FUNCTION_BLOCK PUBLIC WORD_TO_TestSuite EXTENDS TcUnit.FB_TestSuite
VAR
END_VAR

Check_WORD_TO_BOOL_Max();
Check_WORD_TO_BOOL_Min();
Check_WORD_TO_BYTE_Max();
Check_WORD_TO_BYTE_Min();
Check_WORD_TO_BYTE_TooHigh();
Check_WORD_TO_WORD_Max();
Check_WORD_TO_WORD_Min();
Check_WORD_TO_DWORD_Max();
Check_WORD_TO_DWORD_Min();
Check_WORD_TO_LWORD_Max();
Check_WORD_TO_LWORD_Min();
Check_WORD_TO_SINT_Max();
Check_WORD_TO_SINT_Min();
Check_WORD_TO_SINT_TooHigh();
Check_WORD_TO_INT_Max();
Check_WORD_TO_INT_Min();
Check_WORD_TO_INT_TooHigh();
Check_WORD_TO_DINT_Max();
Check_WORD_TO_DINT_Min();
Check_WORD_TO_LINT_Max();
Check_WORD_TO_LINT_Min();
Check_WORD_TO_USINT_Max();
Check_WORD_TO_USINT_Min();
Check_WORD_TO_USINT_TooHigh();
Check_WORD_TO_UINT_Max();
Check_WORD_TO_UINT_Min();
Check_WORD_TO_UDINT_Max();
Check_WORD_TO_UDINT_Min();
Check_WORD_TO_ULINT_Max();
Check_WORD_TO_ULINT_Min();
Check_WORD_TO_REAL_Max();
Check_WORD_TO_REAL_Min();
Check_WORD_TO_LREAL_Max();
Check_WORD_TO_LREAL_Min();
Check_WORD_TO_TIME_Max();
Check_WORD_TO_TIME_Min();
Check_WORD_TO_TOD_Max();
Check_WORD_TO_TOD_Min();
Check_WORD_TO_DATE_Max();
Check_WORD_TO_DATE_Min();
Check_WORD_TO_DT_Max();
Check_WORD_TO_DT_Min();
Check_WORD_TO_STRING_Max();
Check_WORD_TO_STRING_Min();

METHOD PUBLIC Check_WORD_TO_BOOL_Min
VAR
	value : WORD := DatatypeLimits.WORD_MIN_VALUE;
	actual : BOOL;
	converted : BOOL;
	equal : BOOL;
END_VAR
TEST('Check_WORD_TO_BOOL_Min');

// @TEST-RUN
converted := TryConvert_WORD_TO_Destination(value, actual);
equal := actual = WORD_TO_BOOL(value);

// @TEST-ASSERT
AssertTrue(Condition := equal, Message := 'Did not convert WORD to BOOL correctly');
AssertTrue(Condition := converted, Message := 'Did not report WORD to BOOL conversion was successful');

TEST_FINISHED();
END_METHOD

METHOD PUBLIC Check_WORD_TO_BOOL_Max
VAR
	value : WORD := DatatypeLimits.WORD_MAX_VALUE;
	actual : BOOL;
	converted : BOOL;
	equal : BOOL;
END_VAR
TEST('Check_WORD_TO_BOOL_Max');

// @TEST-RUN
converted := TryConvert_WORD_TO_Destination(value, actual);
equal := actual = WORD_TO_BOOL(value);

// @TEST-ASSERT
AssertTrue(Condition := equal, Message := 'Did not convert WORD to BOOL correctly');
AssertTrue(Condition := converted, Message := 'Did not report WORD to BOOL conversion was successful');

TEST_FINISHED();
END_METHOD

METHOD PUBLIC Check_WORD_TO_BYTE_Min
VAR
	value : WORD := DatatypeLimits.WORD_MIN_VALUE;
	actual : BYTE;
	converted : BOOL;
	equal : BOOL;
END_VAR
TEST('Check_WORD_TO_BYTE_Min');

// @TEST-RUN
converted := TryConvert_WORD_TO_Destination(value, actual);
equal := actual = WORD_TO_BYTE(value);

// @TEST-ASSERT
AssertTrue(Condition := equal, Message := 'Did not convert WORD to BYTE correctly');
AssertTrue(Condition := converted, Message := 'Did not report WORD to BYTE conversion was successful');

TEST_FINISHED();
END_METHOD

METHOD PUBLIC Check_WORD_TO_BYTE_TooHigh
VAR
	value : WORD := DatatypeLimits.WORD_MAX_VALUE;
	actual : BYTE;
	converted : BOOL;
END_VAR
TEST('Check_WORD_TO_BYTE_TooHigh');

// @TEST-RUN
converted := TryConvert_WORD_TO_Destination(value, actual);

// @TEST-ASSERT
AssertFalse(Condition := converted, Message := 'Did not report WORD to BYTE conversion was prevented');

TEST_FINISHED();
END_METHOD

METHOD PUBLIC Check_WORD_TO_BYTE_Max
VAR
	value : WORD := DatatypeLimits.MAX_VALUE_OF_WORD_WHICH_CAN_BE_HELD_IN_A_BYTE;
	actual : BYTE;
	converted : BOOL;
	equal : BOOL;
END_VAR
TEST('Check_WORD_TO_BYTE_Max');

// @TEST-RUN
converted := TryConvert_WORD_TO_Destination(value, actual);
equal := actual = WORD_TO_BYTE(value);

// @TEST-ASSERT
AssertTrue(Condition := equal, Message := 'Did not convert WORD to BYTE correctly');
AssertTrue(Condition := converted, Message := 'Did not report WORD to BYTE conversion was successful');

TEST_FINISHED();
END_METHOD

METHOD PUBLIC Check_WORD_TO_DATE_Min
VAR
	value : WORD := DatatypeLimits.WORD_MIN_VALUE;
	actual : DATE;
	converted : BOOL;
	equal : BOOL;
END_VAR
TEST('Check_WORD_TO_DATE_Min');

// @TEST-RUN
converted := TryConvert_WORD_TO_Destination(value, actual);
equal := actual = WORD_TO_DATE(value);

// @TEST-ASSERT
AssertTrue(Condition := equal, Message := 'Did not convert WORD to DATE correctly');
AssertTrue(Condition := converted, Message := 'Did not report WORD to DATE conversion was successful');

TEST_FINISHED();
END_METHOD

METHOD PUBLIC Check_WORD_TO_DATE_Max
VAR
	value : WORD := DatatypeLimits.WORD_MAX_VALUE;
	actual : DATE;
	converted : BOOL;
	equal : BOOL;
END_VAR
TEST('Check_WORD_TO_DATE_Max');

// @TEST-RUN
converted := TryConvert_WORD_TO_Destination(value, actual);
equal := actual = WORD_TO_DATE(value);

// @TEST-ASSERT
AssertTrue(Condition := equal, Message := 'Did not convert WORD to DATE correctly');
AssertTrue(Condition := converted, Message := 'Did not report WORD to DATE conversion was successful');

TEST_FINISHED();
END_METHOD

METHOD PUBLIC Check_WORD_TO_DINT_Min
VAR
	value : WORD := DatatypeLimits.WORD_MIN_VALUE;
	actual : DINT;
	converted : BOOL;
	equal : BOOL;
END_VAR
TEST('Check_WORD_TO_DINT_Min');

// @TEST-RUN
converted := TryConvert_WORD_TO_Destination(value, actual);
equal := actual = WORD_TO_DINT(value);

// @TEST-ASSERT
AssertTrue(Condition := equal, Message := 'Did not convert WORD to DINT correctly');
AssertTrue(Condition := converted, Message := 'Did not report WORD to DINT conversion was successful');

TEST_FINISHED();
END_METHOD

METHOD PUBLIC Check_WORD_TO_DINT_Max
VAR
	value : WORD := DatatypeLimits.WORD_MAX_VALUE;
	actual : DINT;
	converted : BOOL;
	equal : BOOL;
END_VAR
TEST('Check_WORD_TO_DINT_Max');

// @TEST-RUN
converted := TryConvert_WORD_TO_Destination(value, actual);
equal := actual = WORD_TO_DINT(value);

// @TEST-ASSERT
AssertTrue(Condition := equal, Message := 'Did not convert WORD to DINT correctly');
AssertTrue(Condition := converted, Message := 'Did not report WORD to DINT conversion was successful');

TEST_FINISHED();
END_METHOD

METHOD PUBLIC Check_WORD_TO_DT_Min
VAR
	value : WORD := DatatypeLimits.WORD_MIN_VALUE;
	actual : DT;
	converted : BOOL;
	equal : BOOL;
END_VAR
TEST('Check_WORD_TO_DT_Min');

// @TEST-RUN
converted := TryConvert_WORD_TO_Destination(value, actual);
equal := actual = WORD_TO_DT(value);

// @TEST-ASSERT
AssertTrue(Condition := equal, Message := 'Did not convert WORD to DT correctly');
AssertTrue(Condition := converted, Message := 'Did not report WORD to DT conversion was successful');

TEST_FINISHED();
END_METHOD

METHOD PUBLIC Check_WORD_TO_DT_Max
VAR
	value : WORD := DatatypeLimits.WORD_MAX_VALUE;
	actual : DT;
	converted : BOOL;
	equal : BOOL;
END_VAR
TEST('Check_WORD_TO_DT_Max');

// @TEST-RUN
converted := TryConvert_WORD_TO_Destination(value, actual);
equal := actual = WORD_TO_DT(value);

// @TEST-ASSERT
AssertTrue(Condition := equal, Message := 'Did not convert WORD to DT correctly');
AssertTrue(Condition := converted, Message := 'Did not report WORD to DT conversion was successful');

TEST_FINISHED();
END_METHOD

METHOD PUBLIC Check_WORD_TO_DWORD_Min
VAR
	value : WORD := DatatypeLimits.WORD_MIN_VALUE;
	actual : DWORD;
	converted : BOOL;
	equal : BOOL;
END_VAR
TEST('Check_WORD_TO_DWORD_Min');

// @TEST-RUN
converted := TryConvert_WORD_TO_Destination(value, actual);
equal := actual = WORD_TO_DWORD(value);

// @TEST-ASSERT
AssertTrue(Condition := equal, Message := 'Did not convert WORD to DWORD correctly');
AssertTrue(Condition := converted, Message := 'Did not report WORD to DWORD conversion was successful');

TEST_FINISHED();
END_METHOD

METHOD PUBLIC Check_WORD_TO_DWORD_Max
VAR
	value : WORD := DatatypeLimits.WORD_MAX_VALUE;
	actual : DWORD;
	converted : BOOL;
	equal : BOOL;
END_VAR
TEST('Check_WORD_TO_DWORD_Max');

// @TEST-RUN
converted := TryConvert_WORD_TO_Destination(value, actual);
equal := actual = WORD_TO_DWORD(value);

// @TEST-ASSERT
AssertTrue(Condition := equal, Message := 'Did not convert WORD to DWORD correctly');
AssertTrue(Condition := converted, Message := 'Did not report WORD to DWORD conversion was successful');

TEST_FINISHED();
END_METHOD

METHOD PUBLIC Check_WORD_TO_INT_Min
VAR
	value : WORD := DatatypeLimits.WORD_MIN_VALUE;
	actual : INT;
	converted : BOOL;
	equal : BOOL;
END_VAR
TEST('Check_WORD_TO_INT_Min');

// @TEST-RUN
converted := TryConvert_WORD_TO_Destination(value, actual);
equal := actual = WORD_TO_INT(value);

// @TEST-ASSERT
AssertTrue(Condition := equal, Message := 'Did not convert WORD to INT correctly');
AssertTrue(Condition := converted, Message := 'Did not report WORD to INT conversion was successful');

TEST_FINISHED();
END_METHOD

METHOD PUBLIC Check_WORD_TO_INT_TooHigh
VAR
	value : WORD := DatatypeLimits.WORD_MAX_VALUE;
	actual : INT;
	converted : BOOL;
END_VAR
TEST('Check_WORD_TO_INT_TooHigh');

// @TEST-RUN
converted := TryConvert_WORD_TO_Destination(value, actual);

// @TEST-ASSERT
AssertFalse(Condition := converted, Message := 'Did not report WORD to INT conversion was prevented');

TEST_FINISHED();
END_METHOD

METHOD PUBLIC Check_WORD_TO_INT_Max
VAR
	value : WORD := DatatypeLimits.MAX_VALUE_OF_WORD_WHICH_CAN_BE_HELD_IN_A_INT;
	actual : INT;
	converted : BOOL;
	equal : BOOL;
END_VAR
TEST('Check_WORD_TO_INT_Max');

// @TEST-RUN
converted := TryConvert_WORD_TO_Destination(value, actual);
equal := actual = WORD_TO_INT(value);

// @TEST-ASSERT
AssertTrue(Condition := equal, Message := 'Did not convert WORD to INT correctly');
AssertTrue(Condition := converted, Message := 'Did not report WORD to INT conversion was successful');

TEST_FINISHED();
END_METHOD

METHOD PUBLIC Check_WORD_TO_LINT_Min
VAR
	value : WORD := DatatypeLimits.WORD_MIN_VALUE;
	actual : LINT;
	converted : BOOL;
	equal : BOOL;
END_VAR
TEST('Check_WORD_TO_LINT_Min');

// @TEST-RUN
converted := TryConvert_WORD_TO_Destination(value, actual);
equal := actual = WORD_TO_LINT(value);

// @TEST-ASSERT
AssertTrue(Condition := equal, Message := 'Did not convert WORD to LINT correctly');
AssertTrue(Condition := converted, Message := 'Did not report WORD to LINT conversion was successful');

TEST_FINISHED();
END_METHOD

METHOD PUBLIC Check_WORD_TO_LINT_Max
VAR
	value : WORD := DatatypeLimits.WORD_MAX_VALUE;
	actual : LINT;
	converted : BOOL;
	equal : BOOL;
END_VAR
TEST('Check_WORD_TO_LINT_Max');

// @TEST-RUN
converted := TryConvert_WORD_TO_Destination(value, actual);
equal := actual = WORD_TO_LINT(value);

// @TEST-ASSERT
AssertTrue(Condition := equal, Message := 'Did not convert WORD to LINT correctly');
AssertTrue(Condition := converted, Message := 'Did not report WORD to LINT conversion was successful');

TEST_FINISHED();
END_METHOD

METHOD PUBLIC Check_WORD_TO_LREAL_Min
VAR
	value : WORD := DatatypeLimits.WORD_MIN_VALUE;
	actual : LREAL;
	converted : BOOL;
	equal : BOOL;
END_VAR
TEST('Check_WORD_TO_LREAL_Min');

// @TEST-RUN
converted := TryConvert_WORD_TO_Destination(value, actual);
equal := actual = WORD_TO_LREAL(value);

// @TEST-ASSERT
AssertTrue(Condition := equal, Message := 'Did not convert WORD to LREAL correctly');
AssertTrue(Condition := converted, Message := 'Did not report WORD to LREAL conversion was successful');

TEST_FINISHED();
END_METHOD

METHOD PUBLIC Check_WORD_TO_LREAL_Max
VAR
	value : WORD := DatatypeLimits.WORD_MAX_VALUE;
	actual : LREAL;
	converted : BOOL;
	equal : BOOL;
END_VAR
TEST('Check_WORD_TO_LREAL_Max');

// @TEST-RUN
converted := TryConvert_WORD_TO_Destination(value, actual);
equal := actual = WORD_TO_LREAL(value);

// @TEST-ASSERT
AssertTrue(Condition := equal, Message := 'Did not convert WORD to LREAL correctly');
AssertTrue(Condition := converted, Message := 'Did not report WORD to LREAL conversion was successful');

TEST_FINISHED();
END_METHOD

METHOD PUBLIC Check_WORD_TO_LWORD_Min
VAR
	value : WORD := DatatypeLimits.WORD_MIN_VALUE;
	actual : LWORD;
	converted : BOOL;
	equal : BOOL;
END_VAR
TEST('Check_WORD_TO_LWORD_Min');

// @TEST-RUN
converted := TryConvert_WORD_TO_Destination(value, actual);
equal := actual = WORD_TO_LWORD(value);

// @TEST-ASSERT
AssertTrue(Condition := equal, Message := 'Did not convert WORD to LWORD correctly');
AssertTrue(Condition := converted, Message := 'Did not report WORD to LWORD conversion was successful');

TEST_FINISHED();
END_METHOD

METHOD PUBLIC Check_WORD_TO_LWORD_Max
VAR
	value : WORD := DatatypeLimits.WORD_MAX_VALUE;
	actual : LWORD;
	converted : BOOL;
	equal : BOOL;
END_VAR
TEST('Check_WORD_TO_LWORD_Max');

// @TEST-RUN
converted := TryConvert_WORD_TO_Destination(value, actual);
equal := actual = WORD_TO_LWORD(value);

// @TEST-ASSERT
AssertTrue(Condition := equal, Message := 'Did not convert WORD to LWORD correctly');
AssertTrue(Condition := converted, Message := 'Did not report WORD to LWORD conversion was successful');

TEST_FINISHED();
END_METHOD

METHOD PUBLIC Check_WORD_TO_REAL_Min
VAR
	value : WORD := DatatypeLimits.WORD_MIN_VALUE;
	actual : REAL;
	converted : BOOL;
	equal : BOOL;
END_VAR
TEST('Check_WORD_TO_REAL_Min');

// @TEST-RUN
converted := TryConvert_WORD_TO_Destination(value, actual);
equal := actual = WORD_TO_REAL(value);

// @TEST-ASSERT
AssertTrue(Condition := equal, Message := 'Did not convert WORD to REAL correctly');
AssertTrue(Condition := converted, Message := 'Did not report WORD to REAL conversion was successful');

TEST_FINISHED();
END_METHOD

METHOD PUBLIC Check_WORD_TO_REAL_Max
VAR
	value : WORD := DatatypeLimits.WORD_MAX_VALUE;
	actual : REAL;
	converted : BOOL;
	equal : BOOL;
END_VAR
TEST('Check_WORD_TO_REAL_Max');

// @TEST-RUN
converted := TryConvert_WORD_TO_Destination(value, actual);
equal := actual = WORD_TO_REAL(value);

// @TEST-ASSERT
AssertTrue(Condition := equal, Message := 'Did not convert WORD to REAL correctly');
AssertTrue(Condition := converted, Message := 'Did not report WORD to REAL conversion was successful');

TEST_FINISHED();
END_METHOD

METHOD PUBLIC Check_WORD_TO_SINT_Min
VAR
	value : WORD := DatatypeLimits.WORD_MIN_VALUE;
	actual : SINT;
	converted : BOOL;
	equal : BOOL;
END_VAR
TEST('Check_WORD_TO_SINT_Min');

// @TEST-RUN
converted := TryConvert_WORD_TO_Destination(value, actual);
equal := actual = WORD_TO_SINT(value);

// @TEST-ASSERT
AssertTrue(Condition := equal, Message := 'Did not convert WORD to SINT correctly');
AssertTrue(Condition := converted, Message := 'Did not report WORD to SINT conversion was successful');

TEST_FINISHED();
END_METHOD

METHOD PUBLIC Check_WORD_TO_SINT_TooHigh
VAR
	value : WORD := DatatypeLimits.WORD_MAX_VALUE;
	actual : SINT;
	converted : BOOL;
END_VAR
TEST('Check_WORD_TO_SINT_TooHigh');

// @TEST-RUN
converted := TryConvert_WORD_TO_Destination(value, actual);

// @TEST-ASSERT
AssertFalse(Condition := converted, Message := 'Did not report WORD to SINT conversion was prevented');

TEST_FINISHED();
END_METHOD

METHOD PUBLIC Check_WORD_TO_SINT_Max
VAR
	value : WORD := DatatypeLimits.MAX_VALUE_OF_WORD_WHICH_CAN_BE_HELD_IN_A_SINT;
	actual : SINT;
	converted : BOOL;
	equal : BOOL;
END_VAR
TEST('Check_WORD_TO_SINT_Max');

// @TEST-RUN
converted := TryConvert_WORD_TO_Destination(value, actual);
equal := actual = WORD_TO_SINT(value);

// @TEST-ASSERT
AssertTrue(Condition := equal, Message := 'Did not convert WORD to SINT correctly');
AssertTrue(Condition := converted, Message := 'Did not report WORD to SINT conversion was successful');

TEST_FINISHED();
END_METHOD

METHOD PUBLIC Check_WORD_TO_STRING_Min
VAR
	value : WORD := DatatypeLimits.WORD_MIN_VALUE;
	actual : STRING;
	converted : BOOL;
	equal : BOOL;
END_VAR
TEST('Check_WORD_TO_STRING_Min');

// @TEST-RUN
converted := TryConvert_WORD_TO_Destination(value, actual);
equal := actual = WORD_TO_STRING(value);

// @TEST-ASSERT
AssertTrue(Condition := equal, Message := 'Did not convert WORD to STRING correctly');
AssertTrue(Condition := converted, Message := 'Did not report WORD to STRING conversion was successful');

TEST_FINISHED();
END_METHOD

METHOD PUBLIC Check_WORD_TO_STRING_Max
VAR
	value : WORD := DatatypeLimits.WORD_MAX_VALUE;
	actual : STRING;
	converted : BOOL;
	equal : BOOL;
END_VAR
TEST('Check_WORD_TO_STRING_Max');

// @TEST-RUN
converted := TryConvert_WORD_TO_Destination(value, actual);
equal := actual = WORD_TO_STRING(value);

// @TEST-ASSERT
AssertTrue(Condition := equal, Message := 'Did not convert WORD to STRING correctly');
AssertTrue(Condition := converted, Message := 'Did not report WORD to STRING conversion was successful');

TEST_FINISHED();
END_METHOD

METHOD PUBLIC Check_WORD_TO_TIME_Min
VAR
	value : WORD := DatatypeLimits.WORD_MIN_VALUE;
	actual : TIME;
	converted : BOOL;
	equal : BOOL;
END_VAR
TEST('Check_WORD_TO_TIME_Min');

// @TEST-RUN
converted := TryConvert_WORD_TO_Destination(value, actual);
equal := actual = WORD_TO_TIME(value);

// @TEST-ASSERT
AssertTrue(Condition := equal, Message := 'Did not convert WORD to TIME correctly');
AssertTrue(Condition := converted, Message := 'Did not report WORD to TIME conversion was successful');

TEST_FINISHED();
END_METHOD

METHOD PUBLIC Check_WORD_TO_TIME_Max
VAR
	value : WORD := DatatypeLimits.WORD_MAX_VALUE;
	actual : TIME;
	converted : BOOL;
	equal : BOOL;
END_VAR
TEST('Check_WORD_TO_TIME_Max');

// @TEST-RUN
converted := TryConvert_WORD_TO_Destination(value, actual);
equal := actual = WORD_TO_TIME(value);

// @TEST-ASSERT
AssertTrue(Condition := equal, Message := 'Did not convert WORD to TIME correctly');
AssertTrue(Condition := converted, Message := 'Did not report WORD to TIME conversion was successful');

TEST_FINISHED();
END_METHOD

METHOD PUBLIC Check_WORD_TO_TOD_Min
VAR
	value : WORD := DatatypeLimits.WORD_MIN_VALUE;
	actual : TOD;
	converted : BOOL;
	equal : BOOL;
END_VAR
TEST('Check_WORD_TO_TOD_Min');

// @TEST-RUN
converted := TryConvert_WORD_TO_Destination(value, actual);
equal := actual = WORD_TO_TOD(value);

// @TEST-ASSERT
AssertTrue(Condition := equal, Message := 'Did not convert WORD to TOD correctly');
AssertTrue(Condition := converted, Message := 'Did not report WORD to TOD conversion was successful');

TEST_FINISHED();
END_METHOD

METHOD PUBLIC Check_WORD_TO_TOD_Max
VAR
	value : WORD := DatatypeLimits.WORD_MAX_VALUE;
	actual : TOD;
	converted : BOOL;
	equal : BOOL;
END_VAR
TEST('Check_WORD_TO_TOD_Max');

// @TEST-RUN
converted := TryConvert_WORD_TO_Destination(value, actual);
equal := actual = WORD_TO_TOD(value);

// @TEST-ASSERT
AssertTrue(Condition := equal, Message := 'Did not convert WORD to TOD correctly');
AssertTrue(Condition := converted, Message := 'Did not report WORD to TOD conversion was successful');

TEST_FINISHED();
END_METHOD

METHOD PUBLIC Check_WORD_TO_UDINT_Min
VAR
	value : WORD := DatatypeLimits.WORD_MIN_VALUE;
	actual : UDINT;
	converted : BOOL;
	equal : BOOL;
END_VAR
TEST('Check_WORD_TO_UDINT_Min');

// @TEST-RUN
converted := TryConvert_WORD_TO_Destination(value, actual);
equal := actual = WORD_TO_UDINT(value);

// @TEST-ASSERT
AssertTrue(Condition := equal, Message := 'Did not convert WORD to UDINT correctly');
AssertTrue(Condition := converted, Message := 'Did not report WORD to UDINT conversion was successful');

TEST_FINISHED();
END_METHOD

METHOD PUBLIC Check_WORD_TO_UDINT_Max
VAR
	value : WORD := DatatypeLimits.WORD_MAX_VALUE;
	actual : UDINT;
	converted : BOOL;
	equal : BOOL;
END_VAR
TEST('Check_WORD_TO_UDINT_Max');

// @TEST-RUN
converted := TryConvert_WORD_TO_Destination(value, actual);
equal := actual = WORD_TO_UDINT(value);

// @TEST-ASSERT
AssertTrue(Condition := equal, Message := 'Did not convert WORD to UDINT correctly');
AssertTrue(Condition := converted, Message := 'Did not report WORD to UDINT conversion was successful');

TEST_FINISHED();
END_METHOD

METHOD PUBLIC Check_WORD_TO_UINT_Min
VAR
	value : WORD := DatatypeLimits.WORD_MIN_VALUE;
	actual : UINT;
	converted : BOOL;
	equal : BOOL;
END_VAR
TEST('Check_WORD_TO_UINT_Min');

// @TEST-RUN
converted := TryConvert_WORD_TO_Destination(value, actual);
equal := actual = WORD_TO_UINT(value);

// @TEST-ASSERT
AssertTrue(Condition := equal, Message := 'Did not convert WORD to UINT correctly');
AssertTrue(Condition := converted, Message := 'Did not report WORD to UINT conversion was successful');

TEST_FINISHED();
END_METHOD

METHOD PUBLIC Check_WORD_TO_UINT_Max
VAR
	value : WORD := DatatypeLimits.WORD_MAX_VALUE;
	actual : UINT;
	converted : BOOL;
	equal : BOOL;
END_VAR
TEST('Check_WORD_TO_UINT_Max');

// @TEST-RUN
converted := TryConvert_WORD_TO_Destination(value, actual);
equal := actual = WORD_TO_UINT(value);

// @TEST-ASSERT
AssertTrue(Condition := equal, Message := 'Did not convert WORD to UINT correctly');
AssertTrue(Condition := converted, Message := 'Did not report WORD to UINT conversion was successful');

TEST_FINISHED();
END_METHOD

METHOD PUBLIC Check_WORD_TO_ULINT_Min
VAR
	value : WORD := DatatypeLimits.WORD_MIN_VALUE;
	actual : ULINT;
	converted : BOOL;
	equal : BOOL;
END_VAR
TEST('Check_WORD_TO_ULINT_Min');

// @TEST-RUN
converted := TryConvert_WORD_TO_Destination(value, actual);
equal := actual = WORD_TO_ULINT(value);

// @TEST-ASSERT
AssertTrue(Condition := equal, Message := 'Did not convert WORD to ULINT correctly');
AssertTrue(Condition := converted, Message := 'Did not report WORD to ULINT conversion was successful');

TEST_FINISHED();
END_METHOD

METHOD PUBLIC Check_WORD_TO_ULINT_Max
VAR
	value : WORD := DatatypeLimits.WORD_MAX_VALUE;
	actual : ULINT;
	converted : BOOL;
	equal : BOOL;
END_VAR
TEST('Check_WORD_TO_ULINT_Max');

// @TEST-RUN
converted := TryConvert_WORD_TO_Destination(value, actual);
equal := actual = WORD_TO_ULINT(value);

// @TEST-ASSERT
AssertTrue(Condition := equal, Message := 'Did not convert WORD to ULINT correctly');
AssertTrue(Condition := converted, Message := 'Did not report WORD to ULINT conversion was successful');

TEST_FINISHED();
END_METHOD

METHOD PUBLIC Check_WORD_TO_USINT_Min
VAR
	value : WORD := DatatypeLimits.WORD_MIN_VALUE;
	actual : USINT;
	converted : BOOL;
	equal : BOOL;
END_VAR
TEST('Check_WORD_TO_USINT_Min');

// @TEST-RUN
converted := TryConvert_WORD_TO_Destination(value, actual);
equal := actual = WORD_TO_USINT(value);

// @TEST-ASSERT
AssertTrue(Condition := equal, Message := 'Did not convert WORD to USINT correctly');
AssertTrue(Condition := converted, Message := 'Did not report WORD to USINT conversion was successful');

TEST_FINISHED();
END_METHOD

METHOD PUBLIC Check_WORD_TO_USINT_TooHigh
VAR
	value : WORD := DatatypeLimits.WORD_MAX_VALUE;
	actual : USINT;
	converted : BOOL;
END_VAR
TEST('Check_WORD_TO_USINT_TooHigh');

// @TEST-RUN
converted := TryConvert_WORD_TO_Destination(value, actual);

// @TEST-ASSERT
AssertFalse(Condition := converted, Message := 'Did not report WORD to USINT conversion was prevented');

TEST_FINISHED();
END_METHOD

METHOD PUBLIC Check_WORD_TO_USINT_Max
VAR
	value : WORD := DatatypeLimits.MAX_VALUE_OF_WORD_WHICH_CAN_BE_HELD_IN_A_USINT;
	actual : USINT;
	converted : BOOL;
	equal : BOOL;
END_VAR
TEST('Check_WORD_TO_USINT_Max');

// @TEST-RUN
converted := TryConvert_WORD_TO_Destination(value, actual);
equal := actual = WORD_TO_USINT(value);

// @TEST-ASSERT
AssertTrue(Condition := equal, Message := 'Did not convert WORD to USINT correctly');
AssertTrue(Condition := converted, Message := 'Did not report WORD to USINT conversion was successful');

TEST_FINISHED();
END_METHOD

METHOD PUBLIC Check_WORD_TO_WORD_Min
VAR
	value : WORD := DatatypeLimits.WORD_MIN_VALUE;
	actual : WORD;
	converted : BOOL;
	equal : BOOL;
END_VAR
TEST('Check_WORD_TO_WORD_Min');

// @TEST-RUN
converted := TryConvert_WORD_TO_Destination(value, actual);
equal := actual = value;

// @TEST-ASSERT
AssertTrue(Condition := equal, Message := 'Did not convert WORD to WORD correctly');
AssertTrue(Condition := converted, Message := 'Did not report WORD to WORD conversion was successful');

TEST_FINISHED();
END_METHOD

METHOD PUBLIC Check_WORD_TO_WORD_Max
VAR
	value : WORD := DatatypeLimits.WORD_MAX_VALUE;
	actual : WORD;
	converted : BOOL;
	equal : BOOL;
END_VAR
TEST('Check_WORD_TO_WORD_Max');

// @TEST-RUN
converted := TryConvert_WORD_TO_Destination(value, actual);
equal := actual = value;

// @TEST-ASSERT
AssertTrue(Condition := equal, Message := 'Did not convert WORD to WORD correctly');
AssertTrue(Condition := converted, Message := 'Did not report WORD to WORD conversion was successful');

TEST_FINISHED();
END_METHOD

END_FUNCTION_BLOCK

(* stored: Version 1.1.0.1, ProductVersion 3.1.4024.12
   POU WORD_TO_TestSuite: Id {62b61cec-b9d5-4afe-9616-1f1ed6f0a409}, SpecialFunc None
   Method Check_WORD_TO_BOOL_Min: Id {6142438c-d47a-4da9-8d42-6293b4628560}
   Method Check_WORD_TO_BOOL_Max: Id {a288822c-bbe7-4270-bc39-95718ec0b7ad}
   Method Check_WORD_TO_BYTE_Min: Id {3037b4dd-3f7d-4e39-859f-9677bf5817fa}
   Method Check_WORD_TO_BYTE_TooHigh: Id {85a6002a-c0db-4bdf-b969-26e500799f75}
   Method Check_WORD_TO_BYTE_Max: Id {3ef5763f-3543-4ee7-aa3f-8220aaf52d41}
   Method Check_WORD_TO_DATE_Min: Id {bd5cc940-2d37-497a-bdd9-fd0b288dfc23}
   Method Check_WORD_TO_DATE_Max: Id {717a77d1-1fa5-486a-81df-4a498b6bc5fd}
   Method Check_WORD_TO_DINT_Min: Id {099347bb-7c81-4b27-b820-0bfcdf01984b}
   Method Check_WORD_TO_DINT_Max: Id {17e9500d-e7e8-404a-84e6-c5cc56bc3d7a}
   Method Check_WORD_TO_DT_Min: Id {12d5c476-367d-4e40-b7f2-1b5e238ad9a3}
   Method Check_WORD_TO_DT_Max: Id {8fd068de-e7dc-4ac8-9b3b-48c1a03b6ba3}
   Method Check_WORD_TO_DWORD_Min: Id {6664c6ba-1e1b-4d7f-bc2b-c43fe5a26094}
   Method Check_WORD_TO_DWORD_Max: Id {1281df2d-7439-45bb-b557-29bf236e37ed}
   Method Check_WORD_TO_INT_Min: Id {fe637056-9b3c-41a2-a49d-45961ee08c82}
   Method Check_WORD_TO_INT_TooHigh: Id {803762a4-98b0-4c12-8d2e-27e3e62c9d35}
   Method Check_WORD_TO_INT_Max: Id {02610d71-5cef-44cf-8151-130a3200d9ab}
   Method Check_WORD_TO_LINT_Min: Id {74e403d2-2053-4b3f-88b7-8443a369bdad}
   Method Check_WORD_TO_LINT_Max: Id {e914f27d-8ed9-4db6-a994-28c8f2e4cfad}
   Method Check_WORD_TO_LREAL_Min: Id {ba5663d1-f2d1-4307-bd23-3366ed6e9179}
   Method Check_WORD_TO_LREAL_Max: Id {28990a9f-5632-45e1-b8dd-919a455eb985}
   Method Check_WORD_TO_LWORD_Min: Id {bdc543ab-0adb-471e-8c3c-9da809b3e2a7}
   Method Check_WORD_TO_LWORD_Max: Id {ded4d81f-84db-4ed3-87ac-adc36ce70f12}
   Method Check_WORD_TO_REAL_Min: Id {fac6b1e0-c6d2-45f8-b9a9-e79b38a6d7e2}
   Method Check_WORD_TO_REAL_Max: Id {f72d6e25-14b3-4a7d-8d27-a406de0e0f01}
   Method Check_WORD_TO_SINT_Min: Id {bf4b641a-3205-4440-9415-8e2a4096dd79}
   Method Check_WORD_TO_SINT_TooHigh: Id {d6acec3f-851f-48d2-82a6-4c260cc1dc41}
   Method Check_WORD_TO_SINT_Max: Id {8e90d411-10eb-4b81-87be-654c0663adb1}
   Method Check_WORD_TO_STRING_Min: Id {5de9abee-bb43-4ed3-ba22-5560d7489866}
   Method Check_WORD_TO_STRING_Max: Id {774845f7-d7dc-4ae4-bdef-d92b7621725d}
   Method Check_WORD_TO_TIME_Min: Id {c10bfda8-7c18-4688-a3ca-253c8428679c}
   Method Check_WORD_TO_TIME_Max: Id {a992cc1a-c7cb-4478-a255-3d3d4092457c}
   Method Check_WORD_TO_TOD_Min: Id {cdc4720a-4598-428c-842b-8751d7a5c035}
   Method Check_WORD_TO_TOD_Max: Id {40621d38-8f27-4711-87b8-bcf980ad1d49}
   Method Check_WORD_TO_UDINT_Min: Id {f51698f8-c60e-4d37-a2f9-e87b9cb13c03}
   Method Check_WORD_TO_UDINT_Max: Id {f3503da2-004d-4dcf-a824-dbfd32da2d42}
   Method Check_WORD_TO_UINT_Min: Id {9be4c835-dab3-47bf-ab0f-d4d1aac47758}
   Method Check_WORD_TO_UINT_Max: Id {9809e231-e4cb-49f4-904d-e1c47afb4eb6}
   Method Check_WORD_TO_ULINT_Min: Id {17cbecef-02f0-4711-b364-f6ef47a62eb9}
   Method Check_WORD_TO_ULINT_Max: Id {871368b9-a6b3-4afc-921a-ca49afb28994}
   Method Check_WORD_TO_USINT_Min: Id {8e02364b-6598-4599-8dbc-1dfe10e7eff1}
   Method Check_WORD_TO_USINT_TooHigh: Id {07370261-1acf-40c9-bcf5-7507548fa09d}
   Method Check_WORD_TO_USINT_Max: Id {4af528d0-023f-442e-aa06-bbfe3ee4a7ab}
   Method Check_WORD_TO_WORD_Min: Id {3608d9e3-480a-4f3d-b851-da67311b7aa6}
   Method Check_WORD_TO_WORD_Max: Id {136ee5f7-90b3-4bfe-8fd7-bb03144dd6b4} *)
